// TwinCAT 3 PLC project MAIN
// ProgramVersion: 3.1.4024.0
// libraries:
//   CmpBitmapPool, * (System)
//   Tc2_Standard, * (Beckhoff Automation GmbH)
//   Tc2_System, * (Beckhoff Automation GmbH)
//   Tc3_IoLink, * (Beckhoff Automation GmbH)
//   Tc3_Module, * (Beckhoff Automation GmbH)
//   Util, * (System)
//   VisuSymbols,3.5.10.0,System
// project tree:
//   DUTs/ ImagePool.TcIPO (not stored)
//   / GlobalTextList.TcGTLO, PlcTask.TcTTO, Visualisierungsmanager.TcVMO (not stored), VISU_TASK.TcTTO
//   POUs/Grundfunktionen/ OID200DatenLesen.TcPOU, Hydr_Ventil.TcPOU
//   POUs/Unterfunktionen/ Ansteuerung_Ausgaenge.TcPOU, Automatik_Betrieb.TcPOU, Manueller_Betrieb.TcPOU, Meldeleuchte.TcPOU, Referenzfahrt.TcPOU, Warmlauf.TcPOU
//   POUs/ Saegeautomat.TcPOU, MAIN.TcPOU
//   VISUs/ Visualization.TcVIS
// real-time tasks:
//   TASK PlcTask: cycle T#10ms, priority 20, ADS port 350
//   TASK VISU_TASK: cycle T#200000us, priority 30, ADS port 351
// I/O:
//   DEVICE Gerät 5 (EtherCAT), AmsNetId 5.93.150.74.6.1
//     Klemme 2 (EK1100) [EK1100 EtherCAT-Koppler (2A E-Bus)]
//       Klemme 3 (EL6224) [EL6224 (IO Link Master)]
//       Klemme 4 (EL2024) [EL2024 4K. Dig. Ausgang 24V, 2A]
//       Klemme 5 (EL2024) [EL2024 4K. Dig. Ausgang 24V, 2A]
//       Klemme 5 (EL9011) [EL9011 Endklemme]
//   DEVICE Gerät 7 (CX-BK)
//     Box 1 (CX-BK)
// variable links:
//   MAIN/MAIN Instance <-> Device 5 (EtherCAT)/Term 2 (EK1100)/Term 3 (EL6224)
//     PlcTask Inputs/MAIN.Saegeautomat.OID200.ProzessDatenOID200 <-> IO-Link Port1/Port1: process data
//   MAIN/MAIN Instance <-> Device 5 (EtherCAT)/Term 2 (EK1100)/Term 4 (EL2024)
//     PlcTask Outputs/MAIN.Saegeautomat.Ansteuerung_Ausgaenge.OUT_Stammklemmung_Oben_Hoch <-> Channel 1/Output
//     PlcTask Outputs/MAIN.Saegeautomat.Ansteuerung_Ausgaenge.OUT_Stammklemmung_Oben_Runter <-> Channel 2/Output
//     PlcTask Outputs/MAIN.Saegeautomat.Ansteuerung_Ausgaenge.OUT_Stammklemmung_Unten_Hoch <-> Channel 3/Output
//     PlcTask Outputs/MAIN.Saegeautomat.Ansteuerung_Ausgaenge.OUT_Stammklemmung_Unten_Runter <-> Channel 4/Output
//   MAIN/MAIN Instance <-> Device 5 (EtherCAT)/Term 2 (EK1100)/Term 5 (EL2024)
//     PlcTask Outputs/MAIN.Saegeautomat.Ansteuerung_Ausgaenge.OUT_Saege_Heben <-> Channel 1/Output
//     PlcTask Outputs/MAIN.Saegeautomat.Ansteuerung_Ausgaenge.OUT_Saege_Senken <-> Channel 2/Output
//     PlcTask Outputs/MAIN.Saegeautomat.Ansteuerung_Ausgaenge.OUT_Stammklemmung_Unten_Runter <-> Channel 3/Output
//   MAIN/MAIN Instance <-> Device 7 (CX-BK)/Box 1 (CX-BK)
//     PlcTask Inputs/MAIN.Saegeautomat.IN_BetriebsArt_Automatik <-> Term 2 (KL1104)/Channel 3/Eingang
//     PlcTask Inputs/MAIN.Saegeautomat.IN_BetriebsArt_Manuell <-> Term 2 (KL1104)/Channel 4/Eingang
//     PlcTask Inputs/MAIN.Saegeautomat.IN_BetriebsArt_Referenz <-> Term 2 (KL1104)/Channel 1/Eingang
//     PlcTask Inputs/MAIN.Saegeautomat.IN_BetriebsArt_Warmlauf <-> Term 2 (KL1104)/Channel 2/Eingang
//     PlcTask Inputs/MAIN.Saegeautomat.IN_Einfache_Klemmung <-> Term 3 (KL1104)/Channel 4/Eingang
//     PlcTask Inputs/MAIN.Saegeautomat.IN_Endl_Obere_Stammklemmung_Oben <-> Term 7 (KL1104)/Channel 1/Eingang
//     PlcTask Inputs/MAIN.Saegeautomat.IN_Endl_Obere_Stammklemmung_Unten <-> Term 7 (KL1104)/Channel 2/Eingang
//     PlcTask Inputs/MAIN.Saegeautomat.IN_Endl_Saege_Oben <-> Term 8 (KL1104)/Channel 1/Eingang
//     PlcTask Inputs/MAIN.Saegeautomat.IN_Endl_Saege_Unten <-> Term 8 (KL1104)/Channel 2/Eingang
//     PlcTask Inputs/MAIN.Saegeautomat.IN_Endl_Tastschiene <-> Term 9 (KL1104)/Channel 3/Eingang
//     PlcTask Inputs/MAIN.Saegeautomat.IN_Endl_Untere_Stammklemmung_Oben <-> Term 7 (KL1104)/Channel 3/Eingang
//     PlcTask Inputs/MAIN.Saegeautomat.IN_Endl_Untere_Stammklemmung_Unten <-> Term 7 (KL1104)/Channel 4/Eingang
//     PlcTask Inputs/MAIN.Saegeautomat.IN_Endl_Zufuehrer_Hinten <-> Term 9 (KL1104)/Channel 1/Eingang
//     PlcTask Inputs/MAIN.Saegeautomat.IN_Endl_Zufuehrer_Vorne <-> Term 8 (KL1104)/Channel 4/Eingang
//     PlcTask Inputs/MAIN.Saegeautomat.IN_Hydraulik_EIN <-> Term 4 (KL1104)/Channel 2/Eingang
//     PlcTask Inputs/MAIN.Saegeautomat.IN_Kettenoel_nicht_Leer <-> Term 6 (KL1104)/Channel 3/Eingang
//     PlcTask Inputs/MAIN.Saegeautomat.IN_Kettenschmierung_Manuell_EIN <-> Term 6 (KL1104)/Channel 4/Eingang
//     PlcTask Inputs/MAIN.Saegeautomat.IN_Programm_Einzelsatz <-> Term 3 (KL1104)/Channel 3/Eingang
//     PlcTask Inputs/MAIN.Saegeautomat.IN_Saege_EIN <-> Term 4 (KL1104)/Channel 1/Eingang
//     PlcTask Inputs/MAIN.Saegeautomat.IN_Saege_Hoch <-> Term 6 (KL1104)/Channel 1/Eingang
//     PlcTask Inputs/MAIN.Saegeautomat.IN_Saege_Runter <-> Term 6 (KL1104)/Channel 2/Eingang
//     PlcTask Inputs/MAIN.Saegeautomat.IN_Schaltausg_Druckschalter_Obere_Klemmung <-> Term 9 (KL1104)/Channel 2/Eingang
//     PlcTask Inputs/MAIN.Saegeautomat.IN_Schaltausg_Lichtschranke <-> Term 9 (KL1104)/Channel 4/Eingang
//     PlcTask Inputs/MAIN.Saegeautomat.IN_Stammklemmer_Oben_Hoch <-> Term 5 (KL1104)/Channel 1/Eingang
//     PlcTask Inputs/MAIN.Saegeautomat.IN_Stammklemmer_Oben_Runter <-> Term 5 (KL1104)/Channel 2/Eingang
//     PlcTask Inputs/MAIN.Saegeautomat.IN_Stammklemmer_Unten_Hoch <-> Term 5 (KL1104)/Channel 3/Eingang
//     PlcTask Inputs/MAIN.Saegeautomat.IN_Stammklemmer_Unten_Runter <-> Term 5 (KL1104)/Channel 4/Eingang
//     PlcTask Inputs/MAIN.Saegeautomat.IN_Vorposition_Zufuehrer <-> Term 8 (KL1104)/Channel 3/Eingang
//     PlcTask Inputs/MAIN.Saegeautomat.IN_Zufuehrer_Rueck <-> Term 4 (KL1104)/Channel 3/Eingang
//     PlcTask Inputs/MAIN.Saegeautomat.IN_Zufuehrer_Vor <-> Term 4 (KL1104)/Channel 4/Eingang
//     PlcTask Inputs/MAIN.Saegeautomat.IN_Zyklus_Start <-> Term 3 (KL1104)/Channel 1/Eingang
//     PlcTask Inputs/MAIN.Saegeautomat.IN_Zyklus_Stopp <-> Term 3 (KL1104)/Channel 2/Eingang
//     PlcTask Outputs/MAIN.Saegeautomat.Ansteuerung_Ausgaenge.OUT_Kettenschmierung_EIN <-> Term 11 (KL2114)/Channel 1/Ausgang
//     PlcTask Outputs/MAIN.Saegeautomat.Ansteuerung_Ausgaenge.OUT_Saege_EIN <-> Term 12 (KL2114)/Channel 2/Ausgang
//     PlcTask Outputs/MAIN.Saegeautomat.Ansteuerung_Ausgaenge.OUT_Zufuehrer_Antrieb_Rueck <-> Term 10 (KL2114)/Channel 4/Ausgang
//     PlcTask Outputs/MAIN.Saegeautomat.Ansteuerung_Ausgaenge.OUT_Zufuehrer_Antrieb_Vor <-> Term 10 (KL2114)/Channel 3/Ausgang
//     PlcTask Outputs/MAIN.Saegeautomat.OUT_Hydraulikpumpe_EIN <-> Term 10 (KL2114)/Channel 1/Ausgang
//     PlcTask Outputs/MAIN.Saegeautomat.Steuerung_Meldeleuchten.OUT_Meldeleuchte_Gelb <-> Term 11 (KL2114)/Channel 2/Ausgang
//     PlcTask Outputs/MAIN.Saegeautomat.Steuerung_Meldeleuchten.OUT_Meldeleuchte_Gruen <-> Term 11 (KL2114)/Channel 4/Ausgang
//     PlcTask Outputs/MAIN.Saegeautomat.Steuerung_Meldeleuchten.OUT_Meldeleuchte_Rot <-> Term 11 (KL2114)/Channel 3/Ausgang

CONFIGURATION MAIN
    RESOURCE PLC ON TwinCAT3
        TASK PlcTask(INTERVAL := T#10ms, PRIORITY := 20);
        TASK VISU_TASK(INTERVAL := T#200000us, PRIORITY := 30);
        PROGRAM MAIN WITH PlcTask : MAIN;
        PROGRAM VisuElems_Visu_Prg WITH VISU_TASK : VisuElems.Visu_Prg;
    END_RESOURCE
END_CONFIGURATION

// ---- POUs/MAIN.TcPOU
PROGRAM MAIN
VAR
	Saegeautomat : Saegeautomat;
END_VAR

Saegeautomat();

END_PROGRAM

// ---- POUs/Saegeautomat.TcPOU
FUNCTION_BLOCK Saegeautomat
VAR_INPUT
END_VAR
VAR_OUTPUT
END_VAR
VAR
	//Eingänge Bedienung
	//Organisatorisches
	IN_BetriebsArt_Referenz AT %I* : BOOL;
	IN_BetriebsArt_Warmlauf AT %I* : BOOL;
	IN_BetriebsArt_Automatik AT %I* : BOOL;
	IN_BetriebsArt_Manuell AT %I* : BOOL;
	IN_Kein_Notaus AT %I* : BOOL := TRUE;
	IN_Maschine_EIN AT %I* : BOOL := TRUE;
	IN_Hydraulik_EIN AT %I* : BOOL;
	IN_Maschine_AUS AT %I* : BOOL;
	IN_Hydraulik_AUS AT %I* : BOOL;
	//Manuelle Bedienung
	IN_Kettenschmierung_Manuell_EIN AT %I* : BOOL;
	IN_Zufuehrer_Vor AT %I* : BOOL;
	IN_Zufuehrer_Rueck AT %I* : BOOL;
	IN_Stammklemmer_Oben_Hoch AT %I* : BOOL;
	IN_Stammklemmer_Oben_Runter AT %I* : BOOL;
	IN_Stammklemmer_Unten_Hoch AT %I* : BOOL;
	IN_Stammklemmer_Unten_Runter AT %I* : BOOL;
	IN_Saege_EIN AT %I* : BOOL;
	IN_Saege_AUS AT %I* : BOOL;
	IN_Saege_Hoch AT %I* : BOOL;
	IN_Saege_Runter AT %I* : BOOL;
	//Automatikmodus
	IN_Programm_Einzelsatz AT %I* : BOOL;
	IN_Zyklus_Start AT %I* : BOOL;
	IN_Zyklus_Stopp AT %I* : BOOL;
	IN_Einfache_Klemmung AT %I* : BOOL;
	
	
	//Eingänge Sensorik
	//Zuführer
	IN_Endl_Zufuehrer_Hinten AT %I* : BOOL;
	IN_Endl_Zufuehrer_Vorne AT %I* : BOOL;
	IN_Vorposition_Zufuehrer AT %I* : BOOL;
	IOL_Schaltausg_Distanzsensor_Holzende : BOOL; //Über Schaltausgang oder IO-Link Analogdaten?
	IOL_DistanzSensor_Abst : UINT;
	IN_Schaltausg_Lichtschranke AT %I* : BOOL; 
	
	//Stammklemmung Oben
	IN_Endl_Obere_Stammklemmung_Oben AT %I* : BOOL;
	IN_Endl_Obere_Stammklemmung_Unten AT %I* : BOOL;
	IN_Endl_Tastschiene AT %I* : BOOL;
	IN_Schaltausg_Druckschalter_Obere_Klemmung AT %I* : BOOL;
	//Stammklemmung Unten
	IN_Endl_Untere_Stammklemmung_Oben AT %I* : BOOL;
	IN_Endl_Untere_Stammklemmung_Unten AT %I* : BOOL;
	//Säge
	IN_Endl_Saege_Oben AT %I* : BOOL;
	IN_Endl_Saege_Unten AT %I* : BOOL;
	IN_Kettenoel_nicht_Leer AT %I* : BOOL;
	
	//Ausgänge
	//Ausgänge Hydraulik
	
	//Ausgänge Schalten
	OUT_Hydraulikpumpe_EIN AT %Q* : BOOL;
	//Ausgänge Daten
	
	
		
		
	//Interne Merker
	Maschine_EIN : BOOL;
	Hydraulik_EIN : BOOL;
	Referenz_gefahren : BOOL;
	Zyklus_beendet : BOOL;
	busy : BOOL;
	warten : BOOL;
	
	
	Referenzfahrt : Referenzfahrt;
	Warmlauf : Warmlauf;
	Manueller_Betrieb : Manueller_Betrieb;
	Automatikbetrieb : Automatik_Betrieb;
	Steuerung_Meldeleuchten : Meldeleuchte;
	OID200 : OID200DatenLesen;
	Ansteuerung_Ausgaenge : Ansteuerung_Ausgaenge;
	
	P_Flanke_Zyklus_Stopp : R_TRIG;
	P_Flanke_Zyklus_Start : R_TRIG;
	P_Flanke_Maschine_EIN : R_TRIG;
	

	
END_VAR

P_Flanke_Zyklus_Stopp(CLK := NOT IN_Zyklus_Stopp);
P_Flanke_Zyklus_Start(CLK := IN_Zyklus_Start);
P_Flanke_Maschine_EIN(CLK := IN_Maschine_EIN);


IF IN_Kein_Notaus AND IN_Maschine_EIN THEN
	Maschine_EIN := TRUE;
ELSIF NOT IN_Kein_Notaus OR IN_Maschine_AUS THEN
	Maschine_EIN := FALSE;
END_IF

IF Maschine_EIN AND IN_BetriebsArt_Referenz THEN
	Referenzfahrt(
		Kein_Notaus := IN_Kein_Notaus,
		Programm_Einzelsatz := IN_Programm_Einzelsatz,
		Zyklus_Start := P_Flanke_Zyklus_Start.Q,
		SFCInit := P_Flanke_Zyklus_Stopp.Q OR NOT IN_Kein_Notaus,
		SFCTipMode := IN_Programm_Einzelsatz,
		SFCTip := P_Flanke_Zyklus_Start.Q,
		Endl_Saege_Oben := NOT IN_Endl_Saege_Oben,
		Endl_Obere_Stammklemmung_Oben := NOT IN_Endl_Obere_Stammklemmung_Oben,
		Endl_Untere_Stammklemmung_Unten := NOT IN_Endl_Untere_Stammklemmung_Unten,
		Endl_Zufuehrer_Hinten := NOT IN_Endl_Zufuehrer_Hinten,
		busy := busy,
		Referenz_Gefahren := Referenz_gefahren,
		Zyklus_Beendet := Zyklus_beendet);	
END_IF

IF Maschine_EIN AND IN_BetriebsArt_Warmlauf THEN
	Warmlauf();
END_IF

IF Maschine_EIN AND IN_BetriebsArt_Manuell THEN
	Manueller_Betrieb(
		Kein_Notaus:= IN_Kein_Notaus, 
		Hydraulik_EIN:= IN_Hydraulik_EIN, 
		Hydraulik_AUS:= IN_Hydraulik_AUS, 
		Kettenschmierung_Manuell_EIN:= IN_Kettenschmierung_Manuell_EIN, 
		Zufuehrer_Vor:= IN_Zufuehrer_Vor, 
		Zufuehrer_Rueck:= IN_Zufuehrer_Rueck, 
		Stammklemmer_Oben_Hoch:= IN_Stammklemmer_Oben_Hoch, 
		Stammklemmer_Oben_Runter:= IN_Stammklemmer_Oben_Runter, 
		Stammklemmer_Unten_Hoch:= IN_Stammklemmer_Unten_Hoch, 
		Stammklemmer_Unten_Runter:= IN_Stammklemmer_Unten_Runter, 
		Saege_EIN:= IN_Saege_EIN, 
		Saege_AUS:= IN_Saege_AUS, 
		Saege_Hoch:= IN_Saege_Hoch, 
		Saege_Runter:= IN_Saege_Runter, 
		Endl_Zufuehrer_Hinten:= NOT IN_Endl_Zufuehrer_Hinten, 
		Endl_Zufuehrer_Vorne:= NOT IN_Endl_Zufuehrer_Vorne, 
		Vorposition_Zufuehrer:= NOT IN_Vorposition_Zufuehrer,  
		Endl_Obere_Stammklemmung_Oben:= NOT IN_Endl_Obere_Stammklemmung_Oben, 
		Endl_Obere_Stammklemmung_Unten:= NOT IN_Endl_Obere_Stammklemmung_Unten, 
		Endl_Tastschiene:= NOT IN_Endl_Tastschiene, 
		Schaltausg_Druckschalter_Obere_Klemmung:= NOT IN_Schaltausg_Druckschalter_Obere_Klemmung, 
		Endl_Untere_Stammklemmung_Oben:= NOT IN_Endl_Untere_Stammklemmung_Oben, 
		Endl_Untere_Stammklemmung_Unten:= NOT IN_Endl_Untere_Stammklemmung_Unten, 
		Endl_Saege_Oben:= NOT IN_Endl_Saege_Oben, 
		Endl_Saege_Unten:= NOT IN_Endl_Saege_Unten, 
		);
	
END_IF

IF Maschine_EIN AND IN_BetriebsArt_Automatik THEN
	Automatikbetrieb(
	Kein_Notaus:= IN_Kein_Notaus, 
	Zyklus_Start:= IN_Zyklus_Start, 
	Zyklus_Stopp:= NOT IN_Zyklus_Stopp, 
	Einfache_Klemmung := IN_Einfache_Klemmung,
	SFCInit:= not IN_Zyklus_Stopp, 
	SFCTip:= IN_Programm_Einzelsatz AND IN_Zyklus_Start, 
	SFCTipMode:= IN_Programm_Einzelsatz, 
	Endl_Zufuehrer_Hinten:= NOT IN_Endl_Zufuehrer_Hinten, 
	Endl_Zufuehrer_Vorne:= NOT IN_Endl_Zufuehrer_Vorne, 
	Vorposition_Zufuehrer:= NOT IN_Vorposition_Zufuehrer, 
	IOL_Schaltausg_Distanzsensor_Holzende:= NOT IN_Schaltausg_Lichtschranke, 
	IOL_DistanzSensor_Abst:= IOL_DistanzSensor_Abst, 
	Endl_Obere_Stammklemmung_Oben:= NOT IN_Endl_Obere_Stammklemmung_Oben, 
	Endl_Obere_Stammklemmung_Unten:= NOT IN_Endl_Obere_Stammklemmung_Unten, 
	Endl_Tastschiene:= IN_Endl_Tastschiene, 
	Schaltausg_Druckschalter_Obere_Klemmung:= not IN_Schaltausg_Druckschalter_Obere_Klemmung, 
	Endl_Untere_Stammklemmung_Oben:= NOT IN_Endl_Untere_Stammklemmung_Oben, 
	Endl_Untere_Stammklemmung_Unten:= NOT IN_Endl_Untere_Stammklemmung_Unten, 
	Endl_Saege_Oben:= NOT IN_Endl_Saege_Oben, 
	Endl_Saege_Unten:= NOT IN_Endl_Saege_Unten, 
	Warten_Auf_Weiterschalten=> , 
	Warten_auf_Material=> , 
	QStammklemmung_Oben_Hoch=> , 
	QStammklemmung_Oben_Runter=> , 
	QStammklemmung_Unten_Hoch=> , 
	QStammklemmung_Unten_Runter=> , 
	QSaege_Senken=> , 
	QSaege_Heben=> , 
	QHydraulikpumpe_EIN=> , 
	QZufuehrer_Antrieb_vor=> , 
	QZufuehrer_Antrieb_Rueck=> , 
	QSaege_Antrieb_Ein=> , 
	QKettenschmierung_EIN=> , 
	warten:= warten, 
	Hydraulik_EIN:= Hydraulik_EIN, 
	Zyklus_Beendet:= Zyklus_beendet);
END_IF

Ansteuerung_Ausgaenge(
	Saege_Hoch:= Referenzfahrt.Saege_Heben OR Manueller_Betrieb.QSaege_Heben OR Automatikbetrieb.QSaege_Heben, 
	Saege_Runter:= Manueller_Betrieb.QSaege_Senken OR Automatikbetrieb.QSaege_Senken, 
	Stammklemmung_Oben_Hoch:= Referenzfahrt.Stammklemmung_oben_Hoch OR Manueller_Betrieb.QStammklemmung_Oben_Hoch OR Automatikbetrieb.QStammklemmung_Oben_Hoch, 
	Stammklemmung_Oben_Runter:= Manueller_Betrieb.QStammklemmung_Oben_Runter OR Automatikbetrieb.QStammklemmung_Oben_Runter, 
	Stammklemmung_Unten_Hoch:= Manueller_Betrieb.QStammklemmung_Unten_Hoch OR Automatikbetrieb.QStammklemmung_Unten_Hoch,
	Stammklemmung_Unten_Runter:= Referenzfahrt.Stammklemmung_unten_Runter OR Manueller_Betrieb.QStammklemmung_Unten_Runter OR Automatikbetrieb.QStammklemmung_Unten_Runter,
	Saege_EIN := Manueller_Betrieb.QSaege_Antrieb_Ein OR Automatikbetrieb.QSaege_Antrieb_Ein,
	Zufuehrer_Vor := Manueller_Betrieb.QZufuehrer_Antrieb_vor OR Automatikbetrieb.QZufuehrer_Antrieb_vor,
	Zufuehrer_Rueck := Referenzfahrt.Zufuehrer_Zurueck OR Manueller_Betrieb.QZufuehrer_Antrieb_Rueck OR Automatikbetrieb.QZufuehrer_Antrieb_Rueck,
	endl_Zufuehrer_vorne := NOT IN_Endl_Zufuehrer_Vorne,
	endl_Zufuehrer_hinten := NOT IN_Endl_Zufuehrer_Hinten,
	endl_Zufuehrer_Vorpos := NOT IN_Vorposition_Zufuehrer,
	endl_Stammklemmung_Oben_Oben := NOT IN_Endl_Obere_Stammklemmung_Oben,
	endl_Stammklemmung_Oben_Unten := NOT IN_Endl_Obere_Stammklemmung_Unten,
	endl_Stammklemmung_Unten_Oben := NOT IN_Endl_Untere_Stammklemmung_Oben,
	endl_Stammklemmung_Unten_Unten := NOT IN_Endl_Untere_Stammklemmung_Unten,
	endl_Saege_Oben := NOT IN_Endl_Saege_Oben,
	endl_Saege_Unten:= NOT IN_Endl_Saege_Unten,
	kettenschmierung_EIN := Manueller_Betrieb.QKettenschmierung_EIN OR Automatikbetrieb.QSaege_Antrieb_Ein
);

OUT_Hydraulikpumpe_EIN := Manueller_Betrieb.QHydraulikpumpe_EIN OR Automatikbetrieb.QHydraulikpumpe_EIN OR Referenzfahrt.QHydraulik_EIN;

Steuerung_Meldeleuchten(
	Maschine_EIN := Maschine_EIN,
	Referenz_gefahren := Referenz_gefahren,
	Kettenschmierung_nicht_leer := IN_Kettenoel_nicht_Leer,
	Fehler_liegt_an := ,
	Busy := busy,
	Warten_auf_weiterschalten := Referenzfahrt.Warten_Auf_Weiterschalten OR FALSE, //Automatikbetrieb.Warten_Auf_Weiterschalten
	Zyklus_beendet := );


OID200(
 OID200SchaltSignal => IOL_Schaltausg_Distanzsensor_Holzende,
iOID200Dist_zu_Holz => IOL_DistanzSensor_Abst);

END_FUNCTION_BLOCK

// ---- POUs/Unterfunktionen/Referenzfahrt.TcPOU
FUNCTION_BLOCK Referenzfahrt
VAR_INPUT
	//Taster
	Kein_Notaus : BOOL;
	Programm_Einzelsatz : BOOL;
	Zyklus_Start : BOOL;
	Zyklus_Stopp : BOOL;
	//Merker
	SFCInit : BOOL;
	SFCTip : BOOL;
	SFCTipMode : BOOL;
	//Sensoren	
	Endl_Saege_Oben : BOOL;
	Endl_Obere_Stammklemmung_Oben : BOOL;
	Endl_Untere_Stammklemmung_Unten : BOOL;
	Endl_Zufuehrer_Hinten : BOOL;
	
END_VAR
VAR_OUTPUT
	Saege_Heben : BOOL;
	Stammklemmung_oben_Hoch : BOOL;
	Stammklemmung_unten_Runter : BOOL;
	Zufuehrer_Zurueck : BOOL;
	Warten_Auf_Weiterschalten : BOOL;
	QHydraulik_EIN : BOOL;

END_VAR
VAR_IN_OUT
	//Merker
	busy : BOOL;
	
	Referenz_Gefahren : BOOL;
	Zyklus_Beendet : BOOL;
	
END_VAR
VAR
END_VAR

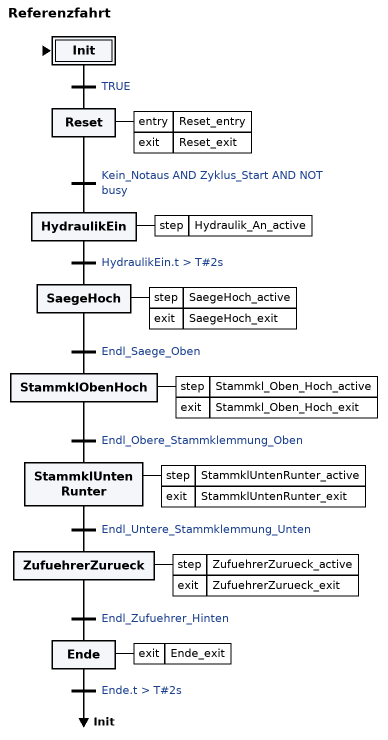
INITIAL_STEP Init:
END_STEP
TRANSITION FROM Init TO Reset
    := TRUE;
END_TRANSITION
STEP Reset:
    Reset_entry(P1);  // entry action
    Reset_exit(P0);  // exit action
END_STEP
TRANSITION FROM Reset TO HydraulikEin
    := Kein_Notaus AND Zyklus_Start AND NOT busy;
END_TRANSITION
STEP HydraulikEin:
    Hydraulik_An_active(N);  // step action
END_STEP
TRANSITION FROM HydraulikEin TO SaegeHoch
    := HydraulikEin.t > T#2s;
END_TRANSITION
STEP SaegeHoch:
    SaegeHoch_active(N);  // step action
    SaegeHoch_exit(P0);  // exit action
END_STEP
TRANSITION FROM SaegeHoch TO StammklObenHoch
    := Endl_Saege_Oben;
END_TRANSITION
STEP StammklObenHoch:
    Stammkl_Oben_Hoch_active(N);  // step action
    Stammkl_Oben_Hoch_exit(P0);  // exit action
END_STEP
TRANSITION FROM StammklObenHoch TO StammklUntenRunter
    := Endl_Obere_Stammklemmung_Oben;
END_TRANSITION
STEP StammklUntenRunter:
    StammklUntenRunter_active(N);  // step action
    StammklUntenRunter_exit(P0);  // exit action
END_STEP
TRANSITION FROM StammklUntenRunter TO ZufuehrerZurueck
    := Endl_Untere_Stammklemmung_Unten;
END_TRANSITION
STEP ZufuehrerZurueck:
    ZufuehrerZurueck_active(N);  // step action
    ZufuehrerZurueck_exit(P0);  // exit action
END_STEP
TRANSITION FROM ZufuehrerZurueck TO Ende
    := Endl_Zufuehrer_Hinten;
END_TRANSITION
STEP Ende:
    Ende_exit(P0);  // exit action
END_STEP
TRANSITION FROM Ende TO Init
    := Ende.t > T#2s;
END_TRANSITION

ACTION Abschluss_active:

END_ACTION

ACTION Ende_exit:
QHydraulik_EIN := FALSE;

busy := FALSE;
Referenz_Gefahren := TRUE;
Zyklus_Beendet := TRUE;
END_ACTION

ACTION Hydraulik_An_active:
QHydraulik_EIN := TRUE;

IF Kein_Notaus AND Zyklus_Start AND NOT busy AND Programm_Einzelsatz THEN 
	Warten_Auf_Weiterschalten := TRUE;
END_IF
END_ACTION

ACTION Hydraulik_An_exit:

END_ACTION

ACTION Reset_entry:
busy := FALSE;
QHydraulik_EIN := FALSE;
Saege_Heben := FALSE;
Stammklemmung_oben_Hoch := FALSE;
Stammklemmung_unten_Runter := FALSE;
Zufuehrer_Zurueck := FALSE;
END_ACTION

ACTION Reset_exit:
busy := TRUE;
Referenz_Gefahren := FALSE;
Zyklus_Beendet := FALSE;

Saege_Heben := FALSE;
Stammklemmung_oben_Hoch := FALSE;
Stammklemmung_unten_Runter := FALSE;
Zufuehrer_Zurueck := FALSE;
END_ACTION

ACTION SaegeHoch_active:
IF NOT Endl_Saege_Oben THEN
	Saege_Heben := TRUE;
END_IF
END_ACTION

ACTION SaegeHoch_exit:
Saege_Heben := FALSE;
END_ACTION

ACTION Stammkl_Oben_Hoch_active:
IF NOT Endl_Obere_Stammklemmung_Oben THEN
	Stammklemmung_oben_Hoch := TRUE;
END_IF
END_ACTION

ACTION Stammkl_Oben_Hoch_exit:
Stammklemmung_oben_Hoch := FALSE;
END_ACTION

ACTION StammklUntenRunter_active:
IF NOT Endl_Untere_Stammklemmung_Unten THEN
	Stammklemmung_unten_Runter := TRUE;
END_IF
END_ACTION

ACTION StammklUntenRunter_exit:
Stammklemmung_unten_Runter := False;
END_ACTION

ACTION ZufuehrerZurueck_active:
IF NOT Endl_Zufuehrer_Hinten THEN
	Zufuehrer_Zurueck := TRUE;
END_IF
END_ACTION

ACTION ZufuehrerZurueck_exit:
Zufuehrer_Zurueck := FALSE;
END_ACTION

END_FUNCTION_BLOCK

// ---- POUs/Unterfunktionen/Warmlauf.TcPOU
FUNCTION_BLOCK Warmlauf
VAR_INPUT
END_VAR
VAR_OUTPUT
END_VAR
VAR
	
END_VAR

END_FUNCTION_BLOCK

// ---- POUs/Unterfunktionen/Manueller_Betrieb.TcPOU
FUNCTION_BLOCK Manueller_Betrieb
VAR_INPUT
	Kein_Notaus : BOOL;
	//Taster auf Bedienfeld
	Hydraulik_EIN : BOOL;
	Hydraulik_AUS : BOOL;
	Kettenschmierung_Manuell_EIN : BOOL;
	Zufuehrer_Vor : BOOL;
	Zufuehrer_Rueck : BOOL;
	Stammklemmer_Oben_Hoch : BOOL;
	Stammklemmer_Oben_Runter : BOOL;
	Stammklemmer_Unten_Hoch : BOOL;
	Stammklemmer_Unten_Runter : BOOL;
	Saege_EIN : BOOL;
	Saege_AUS : BOOL;
	Saege_Hoch : BOOL;
	Saege_Runter : BOOL;
	
	
	//Eingänge Sensorik
	//Zuführer
	Endl_Zufuehrer_Hinten : BOOL;
	Endl_Zufuehrer_Vorne : BOOL;
	Vorposition_Zufuehrer : BOOL;
	//Stammklemmung Oben
	Endl_Obere_Stammklemmung_Oben : BOOL;
	Endl_Obere_Stammklemmung_Unten : BOOL;
	Endl_Tastschiene : BOOL;
	Schaltausg_Druckschalter_Obere_Klemmung : BOOL;
	//Stammklemmung Unten
	Endl_Untere_Stammklemmung_Oben : BOOL;
	Endl_Untere_Stammklemmung_Unten : BOOL;
	//Säge
	Endl_Saege_Oben : BOOL;
	Endl_Saege_Unten : BOOL;
END_VAR
VAR_OUTPUT
	//Ausgänge Hydraulik
	QStammklemmung_Oben_Hoch : BOOL;
	QStammklemmung_Oben_Runter : BOOL;
	QStammklemmung_Unten_Hoch : BOOL;
	QStammklemmung_Unten_Runter : BOOL;
	QSaege_Senken : BOOL;
	QSaege_Heben : BOOL;
	//Ausgänge Schalten
	QHydraulikpumpe_EIN : BOOL;
	QZufuehrer_Antrieb_vor : BOOL;
	QZufuehrer_Antrieb_Rueck : BOOL;
	QSaege_Antrieb_Ein : BOOL;
	QKettenschmierung_EIN : BOOL;
	//Ausgänge Daten
	//FU DATEN
END_VAR
VAR_IN_OUT
	
	
END_VAR
VAR
	Impulsgeber : BLINK;
	TON_Timer_Impuls : TON;
	TON_Timer_Pause : TON;
	Impuls_Zeit : TIME := T#3S;
	Pause_Zeit : TIME := T#3S;
	Impuls : BOOL;
END_VAR

QStammklemmung_Oben_Hoch :=
QStammklemmung_Oben_Runter := 
QStammklemmung_Unten_Hoch := 
QStammklemmung_Unten_Runter := 
QSaege_Senken := 
QSaege_Heben := 
QZufuehrer_Antrieb_vor := 
QZufuehrer_Antrieb_Rueck := 
QSaege_Antrieb_Ein := 
QKettenschmierung_EIN := FALSE;

QHydraulikpumpe_EIN := Hydraulik_EIN;

//Funktionen mit Hydraulik
IF QHydraulikpumpe_EIN THEN
	QStammklemmung_Oben_Hoch := Stammklemmer_Oben_Hoch AND NOT Stammklemmer_Oben_Runter;
	QStammklemmung_Oben_Runter := Stammklemmer_Oben_Runter AND NOT Stammklemmer_Oben_Hoch;
	QStammklemmung_Unten_Hoch := Stammklemmer_Unten_Hoch AND NOT Stammklemmer_Unten_Runter;
	QStammklemmung_Unten_Runter := Stammklemmer_Unten_Runter AND NOT Stammklemmer_Unten_Hoch;
	QSaege_Senken := Saege_Runter AND NOT Saege_Hoch AND NOT Saege_Hoch;
	QSaege_Heben := Saege_Hoch AND NOT Saege_Runter AND NOT Saege_Runter;
END_IF

//Funktionen ohne Hydraulik
IF Hydraulik_EIN THEN
	QHydraulikpumpe_EIN := TRUE;
ELSIF Hydraulik_AUS THEN
	QHydraulikpumpe_EIN := FALSE;
END_IF

QZufuehrer_Antrieb_vor := Zufuehrer_Vor AND NOT Zufuehrer_Rueck;
QZufuehrer_Antrieb_Rueck := Zufuehrer_Rueck AND NOT Zufuehrer_Vor;

QSaege_Antrieb_Ein := Saege_EIN;

Impulsgeber(
	ENABLE := Kettenschmierung_Manuell_EIN,
	TIMELOW := Pause_Zeit,
	TIMEHIGH := Impuls_Zeit,
	OUT => Impuls);

QKettenschmierung_EIN := Kettenschmierung_Manuell_EIN AND Impuls;

END_FUNCTION_BLOCK

// ---- POUs/Unterfunktionen/Automatik_Betrieb.TcPOU
FUNCTION_BLOCK Automatik_Betrieb
VAR_INPUT
	Kein_Notaus : BOOL;
	Zyklus_Start : BOOL;
	Zyklus_Stopp : BOOL;
	SFCInit : BOOL;
	SFCTip : BOOL;
	SFCTipMode : BOOL;
	Einfache_Klemmung : BOOL;
	
	//Eingänge Sensorik
	//Zuführer
	Endl_Zufuehrer_Hinten : BOOL;
	Endl_Zufuehrer_Vorne : BOOL;
	Vorposition_Zufuehrer : BOOL;
	IOL_Schaltausg_Distanzsensor_Holzende : BOOL; //Über Schaltausgang oder IO-Link Analogdaten?
	IOL_DistanzSensor_Abst : UINT;
	//Stammklemmung Oben
	Endl_Obere_Stammklemmung_Oben : BOOL;
	Endl_Obere_Stammklemmung_Unten : BOOL;
	Endl_Tastschiene : BOOL;
	Schaltausg_Druckschalter_Obere_Klemmung : BOOL;
	//Stammklemmung Unten
	Endl_Untere_Stammklemmung_Oben : BOOL;
	Endl_Untere_Stammklemmung_Unten : BOOL;
	//Säge
	Endl_Saege_Oben : BOOL;
	Endl_Saege_Unten : BOOL;
	
END_VAR
VAR_OUTPUT
	Warten_Auf_Weiterschalten :BOOL;
	Warten_auf_Material : BOOL;
	//Hydraulik
	QStammklemmung_Oben_Hoch : BOOL;
	QStammklemmung_Oben_Runter : BOOL;
	QStammklemmung_Unten_Hoch : BOOL;
	QStammklemmung_Unten_Runter : BOOL;
	QSaege_Senken : BOOL;
	QSaege_Heben : BOOL;
	//Ausgänge Schalten
	QHydraulikpumpe_EIN : BOOL;
	QZufuehrer_Antrieb_vor : BOOL;
	QZufuehrer_Antrieb_Rueck : BOOL;
	QSaege_Antrieb_Ein : BOOL;
	QKettenschmierung_EIN : BOOL;
	
END_VAR
VAR_IN_OUT
	warten : BOOL;
	Hydraulik_EIN : BOOL;
	Zyklus_Beendet : BOOL;
END_VAR
VAR
	Holz_Fertig : BOOL;
	Holz_Geklemmt : BOOL;
END_VAR

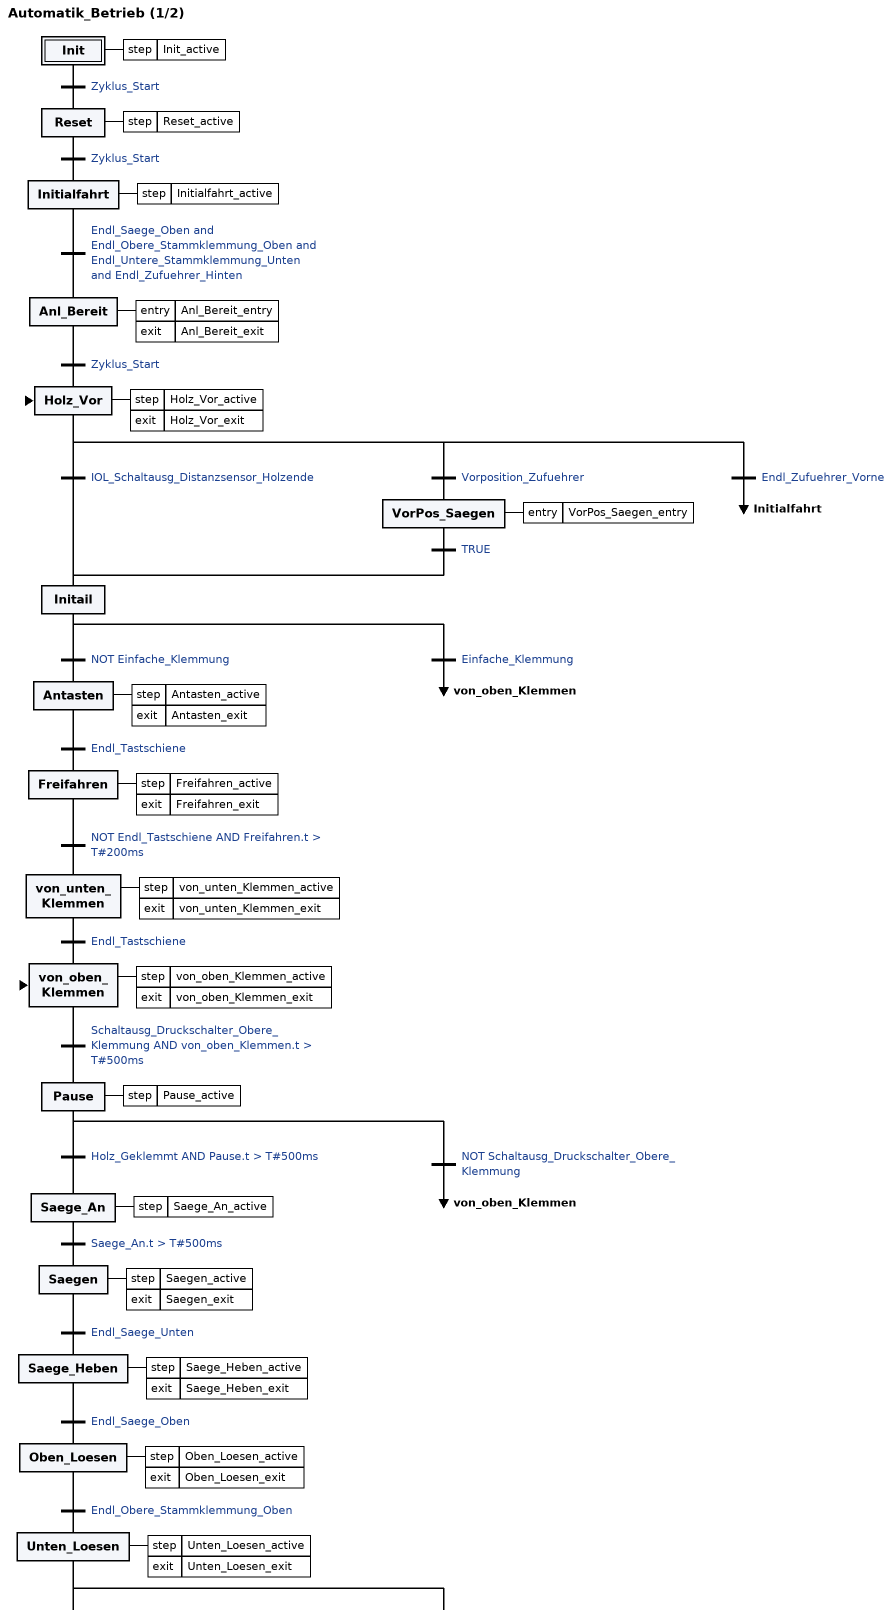
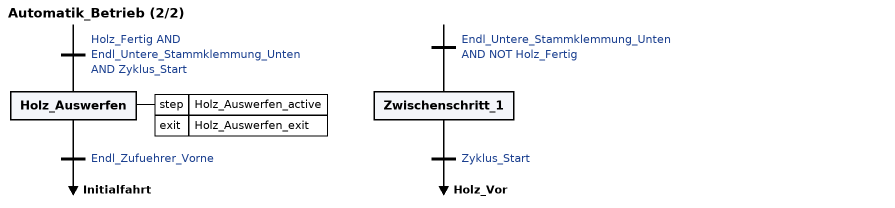
INITIAL_STEP Init:
    Init_active(N);  // step action
END_STEP
TRANSITION FROM Init TO Reset
    := Zyklus_Start;
END_TRANSITION
STEP Reset:
    Reset_active(N);  // step action
END_STEP
TRANSITION FROM Reset TO Initialfahrt_
    := Zyklus_Start;
END_TRANSITION
STEP Initialfahrt_:  // name as stored: Initialfahrt 
    Initialfahrt_active(N);  // step action
END_STEP
TRANSITION FROM Initialfahrt_ TO Anl_Bereit
    := Endl_Saege_Oben and Endl_Obere_Stammklemmung_Oben and Endl_Untere_Stammklemmung_Unten and Endl_Zufuehrer_Hinten;
END_TRANSITION
STEP Anl_Bereit:
    Anl_Bereit_entry(P1);  // entry action
    Anl_Bereit_exit(P0);  // exit action
END_STEP
TRANSITION FROM Anl_Bereit TO Holz_Vor
    := Zyklus_Start;
END_TRANSITION
STEP Holz_Vor:
    Holz_Vor_active(N);  // step action
    Holz_Vor_exit(P0);  // exit action
END_STEP
TRANSITION FROM Holz_Vor TO Initail
    := IOL_Schaltausg_Distanzsensor_Holzende;
END_TRANSITION
TRANSITION FROM Holz_Vor TO VorPos_Saegen
    := Vorposition_Zufuehrer;
END_TRANSITION
STEP VorPos_Saegen:
    VorPos_Saegen_entry(P1);  // entry action
END_STEP
TRANSITION FROM VorPos_Saegen TO Initail
    := TRUE;
END_TRANSITION
TRANSITION FROM Holz_Vor TO Initialfahrt
    := Endl_Zufuehrer_Vorne;
END_TRANSITION
// macro Holz_Klemmen begins
STEP Initail:
END_STEP
TRANSITION FROM Initail TO Antasten
    := NOT Einfache_Klemmung;
END_TRANSITION
STEP Antasten:
    Antasten_active(N);  // step action
    Antasten_exit(P0);  // exit action
END_STEP
TRANSITION FROM Initail TO von_oben_Klemmen
    := Einfache_Klemmung;
END_TRANSITION
TRANSITION FROM Antasten TO Freifahren
    := Endl_Tastschiene;
END_TRANSITION
STEP Freifahren:
    Freifahren_active(N);  // step action
    Freifahren_exit(P0);  // exit action
END_STEP
TRANSITION FROM Freifahren TO von_unten_Klemmen
    := NOT Endl_Tastschiene AND Freifahren.t > T#200ms;
END_TRANSITION
STEP von_unten_Klemmen:
    von_unten_Klemmen_active(N);  // step action
    von_unten_Klemmen_exit(P0);  // exit action
END_STEP
TRANSITION FROM von_unten_Klemmen TO von_oben_Klemmen
    := Endl_Tastschiene;
END_TRANSITION
STEP von_oben_Klemmen:
    von_oben_Klemmen_active(N);  // step action
    von_oben_Klemmen_exit(P0);  // exit action
END_STEP
TRANSITION FROM von_oben_Klemmen TO Pause
    := Schaltausg_Druckschalter_Obere_Klemmung AND von_oben_Klemmen.t > T#500ms;
END_TRANSITION
STEP Pause:
    Pause_active(N);  // step action
END_STEP
TRANSITION FROM Pause TO Saege_An
    := Holz_Geklemmt AND Pause.t > T#500ms;
END_TRANSITION
TRANSITION FROM Pause TO von_oben_Klemmen
    := NOT Schaltausg_Druckschalter_Obere_Klemmung;
END_TRANSITION
// macro Holz_Saegen begins
STEP Saege_An:
    Saege_An_active(N);  // step action
END_STEP
TRANSITION FROM Saege_An TO Saegen
    := Saege_An.t > T#500ms;
END_TRANSITION
STEP Saegen:
    Saegen_active(N);  // step action
    Saegen_exit(P0);  // exit action
END_STEP
TRANSITION FROM Saegen TO Saege_Heben
    := Endl_Saege_Unten;
END_TRANSITION
STEP Saege_Heben:
    Saege_Heben_active(N);  // step action
    Saege_Heben_exit(P0);  // exit action
END_STEP
TRANSITION FROM Saege_Heben TO Oben_Loesen
    := Endl_Saege_Oben;
END_TRANSITION
// macro Holz_Klemmung_Loesen begins
STEP Oben_Loesen:
    Oben_Loesen_active(N);  // step action
    Oben_Loesen_exit(P0);  // exit action
END_STEP
TRANSITION FROM Oben_Loesen TO Unten_Loesen
    := Endl_Obere_Stammklemmung_Oben;
END_TRANSITION
STEP Unten_Loesen:
    Unten_Loesen_active(N);  // step action
    Unten_Loesen_exit(P0);  // exit action
END_STEP
TRANSITION FROM Unten_Loesen TO Holz_Auswerfen
    := Holz_Fertig AND Endl_Untere_Stammklemmung_Unten AND Zyklus_Start;
END_TRANSITION
STEP Holz_Auswerfen:
    Holz_Auswerfen_active(N);  // step action
    Holz_Auswerfen_exit(P0);  // exit action
END_STEP
TRANSITION FROM Holz_Auswerfen TO Initialfahrt
    := Endl_Zufuehrer_Vorne;
END_TRANSITION
TRANSITION FROM Unten_Loesen TO Zwischenschritt_1
    := Endl_Untere_Stammklemmung_Unten AND NOT Holz_Fertig;
END_TRANSITION
STEP Zwischenschritt_1:
END_STEP
TRANSITION FROM Zwischenschritt_1 TO Holz_Vor
    := Zyklus_Start;
END_TRANSITION

ACTION Anl_Bereit_entry:
Warten_auf_Material := TRUE;
QHydraulikpumpe_EIN := FALSE;
END_ACTION

ACTION Anl_Bereit_exit:
Warten_auf_Material := FALSE;
QHydraulikpumpe_EIN := TRUE;
END_ACTION

ACTION Antasten_active:
QStammklemmung_Oben_Runter := TRUE;
END_ACTION

ACTION Antasten_exit:
QStammklemmung_Oben_Runter := FALSE;
END_ACTION

ACTION Freifahren_active:
QStammklemmung_Oben_Hoch := TRUE;
END_ACTION

ACTION Freifahren_exit:
QStammklemmung_Oben_Hoch := FALSE;
END_ACTION

ACTION Holz_Auswerfen_active:
QZufuehrer_Antrieb_vor := TRUE;
END_ACTION

ACTION Holz_Auswerfen_exit:
QZufuehrer_Antrieb_vor := FALSE;
Holz_Fertig := FALSE;
END_ACTION

ACTION Holz_Vor_active:
IF NOT Vorposition_Zufuehrer AND NOT Endl_Zufuehrer_Vorne THEN
	QZufuehrer_Antrieb_vor := TRUE;
END_IF 


IF Vorposition_Zufuehrer OR Endl_Zufuehrer_Vorne OR IOL_Schaltausg_Distanzsensor_Holzende THEN
	QZufuehrer_Antrieb_vor := FALSE;
END_IF
END_ACTION

ACTION Holz_Vor_exit:
QZufuehrer_Antrieb_vor := FALSE;
END_ACTION

ACTION Init_active:
QStammklemmung_Oben_Hoch := 
QStammklemmung_Oben_Runter := 
QStammklemmung_Unten_Hoch := 
QStammklemmung_Unten_Runter := 
QSaege_Senken := 
QSaege_Heben := 
//Ausgänge Schalten
QHydraulikpumpe_EIN := 
QZufuehrer_Antrieb_vor := 
QZufuehrer_Antrieb_Rueck := 
QSaege_Antrieb_Ein := 
QKettenschmierung_EIN := 
Warten_Auf_Weiterschalten :=
Zyklus_Beendet := FALSE;
END_ACTION

ACTION Initialfahrt_active:
IF NOT Endl_Saege_Oben THEN
	QSaege_Heben := TRUE;
	warten := TRUE;
ELSE 
	QSaege_Heben := FALSE;
	warten := FALSE;
END_IF

IF NOT Endl_Obere_Stammklemmung_Oben AND NOT warten THEN
	QStammklemmung_Oben_Hoch := TRUE;
	warten := TRUE;
ELSE
	QStammklemmung_Oben_Hoch := FALSE;
	warten := FALSE;
END_IF

IF NOT Endl_Untere_Stammklemmung_Unten AND NOT warten THEN 
	QStammklemmung_Unten_Runter := TRUE;
	warten := TRUE;
ELSE 
	QStammklemmung_Unten_Runter := FALSE;
	warten := FALSE;
END_IF

IF NOT Endl_Zufuehrer_Hinten THEN
	QZufuehrer_Antrieb_Rueck := TRUE;
ELSE 
	QZufuehrer_Antrieb_Rueck := FALSE;
END_IF
END_ACTION

ACTION Oben_Loesen_active:
QStammklemmung_Oben_Hoch := TRUE;
END_ACTION

ACTION Oben_Loesen_exit:
QStammklemmung_Oben_Hoch := FALSE;
END_ACTION

ACTION Pause_active:
Holz_Geklemmt := TRUE;
END_ACTION

ACTION Reset_active:
//Hydraulik
QStammklemmung_Oben_Hoch := 
QStammklemmung_Oben_Runter := 
QStammklemmung_Unten_Hoch := 
QStammklemmung_Unten_Runter := 
QSaege_Senken := 
QSaege_Heben := 
//Ausgänge Schalten
QHydraulikpumpe_EIN := 
QZufuehrer_Antrieb_vor := 
QZufuehrer_Antrieb_Rueck := 
QSaege_Antrieb_Ein := 
QKettenschmierung_EIN := 
Warten_Auf_Weiterschalten :=
Zyklus_Beendet := FALSE;

QHydraulikpumpe_EIN := TRUE;
END_ACTION

ACTION Saege_An_active:
QSaege_Antrieb_Ein := TRUE;
END_ACTION

ACTION Saege_Heben_active:
QSaege_Heben := TRUE;
END_ACTION

ACTION Saege_Heben_exit:
QSaege_Heben := FALSE;
QSaege_Antrieb_Ein := FALSE;
END_ACTION

ACTION Saegen_active:
QSaege_Senken := TRUE;
END_ACTION

ACTION Saegen_exit:
QSaege_Senken := FALSE;
END_ACTION

ACTION Unten_Loesen_active:
QStammklemmung_Unten_Runter := TRUE;
END_ACTION

ACTION Unten_Loesen_exit:
QStammklemmung_Unten_Runter := FALSE;
END_ACTION

ACTION von_oben_Klemmen_active:
QStammklemmung_Oben_Runter := TRUE;
END_ACTION

ACTION von_oben_Klemmen_exit:
QStammklemmung_Oben_Runter := FALSE;
END_ACTION

ACTION von_unten_Klemmen_active:
QStammklemmung_Unten_Hoch := TRUE;
END_ACTION

ACTION von_unten_Klemmen_exit:
QStammklemmung_Unten_Hoch := FALSE;
END_ACTION

ACTION VorPos_Saegen_entry:
Holz_Fertig := True;
END_ACTION

END_FUNCTION_BLOCK

// ---- POUs/Unterfunktionen/Meldeleuchte.TcPOU
FUNCTION_BLOCK Meldeleuchte
VAR_INPUT
	Zyklus_beendet : BOOL;
	Maschine_EIN : BOOL;
	Fehler_liegt_an : BOOL;
	Kettenschmierung_nicht_leer : BOOL;
	Busy : BOOL;
	Warten_auf_weiterschalten : BOOL;
	Warten_auf_Material : BOOL;
	Referenz_gefahren : BOOL;
	
END_VAR
VAR_OUTPUT
	OUT_Meldeleuchte_Rot AT %Q* : BOOL;//Rot Leuchten: Fehler, Rot Blinken: Kettenöl leer
	OUT_Meldeleuchte_Gelb AT %Q* : BOOL;//Gelb Leuchten:Referenz fehlt, Gelb Blinken: Zyklus beendet
	OUT_Meldeleuchte_Gruen AT %Q* : BOOL;//Grün Leuchten: Zyklus läuft, Grün Blinken: Zyklus läuft(warten auf weiterschalten)
	
END_VAR
VAR
	Impulsgeber : BLINK;
	TON_Timer_Impuls : TON;
	TON_Timer_Pause : TON;
	Impuls_Zeit : TIME := T#500MS;
	Pause_Zeit : TIME := T#500MS;
	Impuls : BOOL;
END_VAR

OUT_Meldeleuchte_Rot := OUT_Meldeleuchte_Gelb := OUT_Meldeleuchte_Gruen := FALSE;

Impulsgeber(
	ENABLE := TRUE,
	TIMELOW := Pause_Zeit,
	TIMEHIGH := Impuls_Zeit,
	OUT => Impuls);

IF Maschine_EIN AND NOT Referenz_gefahren THEN
	OUT_Meldeleuchte_Gelb := TRUE;
ELSIF Maschine_EIN AND Zyklus_beendet THEN
	OUT_Meldeleuchte_Gelb := Impuls;
END_IF

IF Maschine_EIN AND Fehler_liegt_an THEN
	OUT_Meldeleuchte_Rot := TRUE;
ELSIF Maschine_EIN AND NOT Fehler_liegt_an AND NOT Kettenschmierung_nicht_leer THEN
	OUT_Meldeleuchte_Rot := Impuls;
END_IF

IF Maschine_EIN AND Busy AND NOT Warten_auf_weiterschalten THEN 
	OUT_Meldeleuchte_Gruen := TRUE;
ELSIF Maschine_EIN AND Busy AND Warten_auf_weiterschalten THEN
	OUT_Meldeleuchte_Gruen := Impuls;
END_IF

END_FUNCTION_BLOCK

// ---- POUs/Grundfunktionen/OID200DatenLesen.TcPOU
FUNCTION_BLOCK OID200DatenLesen
VAR_INPUT
END_VAR
VAR_OUTPUT
	
	iOID200Dist_zu_Holz : UINT;
	OID200SchaltSignal : BOOL;
	
END_VAR
VAR
	
	ProzessDatenOID200 AT %I* : ARRAY[0..1] OF BYTE;
	ProzessdatenWortOID200 : WORD;
	
END_VAR

ProzessDatenWortOID200 := BYTE_TO_WORD(ProzessdatenOID200[1]) OR SHL(BYTE_TO_WORD(ProzessdatenOID200[0]), 8);
iOID200Dist_zu_Holz := WORD_TO_UINT(SHR(ProzessdatenWortOID200, 4));
OID200SchaltSignal := ProzessDatenOID200[1].0;

END_FUNCTION_BLOCK

// ---- POUs/Unterfunktionen/Ansteuerung_Ausgaenge.TcPOU
FUNCTION_BLOCK Ansteuerung_Ausgaenge
VAR_INPUT
	Saege_Hoch : BOOL;
	Saege_Runter : BOOL;
	Stammklemmung_Oben_Hoch : BOOL;
	Stammklemmung_Oben_Runter : BOOL;
	Stammklemmung_Unten_Hoch : BOOL;
	Stammklemmung_Unten_Runter : BOOL;
	Saege_EIN: BOOL;
	Zufuehrer_Vor : BOOL;
	Zufuehrer_Rueck : BOOL;
	endl_Zufuehrer_vorne : BOOL;
	endl_Zufuehrer_hinten : BOOL;
	endl_Zufuehrer_Vorpos : BOOL;
	endl_Stammklemmung_Oben_Oben : BOOL;
	endl_Stammklemmung_Oben_Unten : BOOL;
	endl_Stammklemmung_Unten_Oben : BOOL;
	endl_Stammklemmung_Unten_Unten : BOOL;
	endl_Saege_Oben : BOOL;
	endl_Saege_Unten : BOOL;
	kettenschmierung_EIN : BOOL;
	
END_VAR
VAR_OUTPUT
	OUT_Saege_Senken AT %Q* : BOOL;
	OUT_Saege_Heben AT %Q* : BOOL;
	OUT_Stammklemmung_Oben_Hoch AT %Q* : BOOL;
	OUT_Stammklemmung_Oben_Runter AT %Q* : BOOL;
	OUT_Stammklemmung_Unten_Hoch AT %Q* : BOOL;
	OUT_Stammklemmung_Unten_Runter AT %Q* : BOOL;
	OUT_Saege_EIN AT %Q* : BOOL;
	OUT_Zufuehrer_Antrieb_Vor AT %Q* : BOOL;
	OUT_Zufuehrer_Antrieb_Rueck AT %Q* : BOOL;
	OUT_Zufuehrer_Antrieb_Enable AT %Q* : BOOL;
	OUT_Kettenschmierung_EIN AT %Q* : BOOL;
END_VAR
VAR
	Saege : Hydr_Ventil;
	Stammklemmung_Oben : Hydr_Ventil;
	Stammklemmung_unten : Hydr_Ventil;
END_VAR


Saege(
	Funktion_A:= Saege_Hoch AND NOT endl_Saege_Oben, 
	Funktion_B:= Saege_Runter AND NOT endl_Saege_Unten, 
	Andere_Ventile_in_Ruhestellung:= Stammklemmung_Oben.Ruhestellung AND Stammklemmung_unten.Ruhestellung, 
	OUT_Spule_A=> OUT_Saege_Heben, 
	OUT_Spule_B=> OUT_Saege_Senken, 
	Status_Invalide=> , 
	Warte_auf_anderes_Ventil=> );

OUT_Saege_EIN := Saege_EIN;
OUT_Kettenschmierung_EIN := kettenschmierung_EIN;
	
Stammklemmung_Oben(
	Funktion_A:= Stammklemmung_Oben_Hoch AND NOT endl_Stammklemmung_Oben_Oben, 
	Funktion_B:= Stammklemmung_Oben_Runter AND NOT endl_Stammklemmung_Oben_Unten, 
	Andere_Ventile_in_Ruhestellung:= Saege.Ruhestellung AND Stammklemmung_unten.Ruhestellung, 
	OUT_Spule_A=> OUT_Stammklemmung_Oben_Hoch, 
	OUT_Spule_B=> OUT_Stammklemmung_Oben_Runter, 
	Status_Invalide=> , 
	Warte_auf_anderes_Ventil=> );
	
Stammklemmung_unten(
	Funktion_A:= Stammklemmung_Unten_Hoch AND NOT endl_Stammklemmung_Unten_Oben, 
	Funktion_B:= Stammklemmung_Unten_Runter AND NOT endl_Stammklemmung_Unten_Unten, 
	Andere_Ventile_in_Ruhestellung:= Saege.Ruhestellung AND Stammklemmung_Oben.Ruhestellung, 
	OUT_Spule_A=> OUT_Stammklemmung_Unten_Hoch, 
	OUT_Spule_B=> OUT_Stammklemmung_Unten_Runter, 
	Status_Invalide=> ,  
	Warte_auf_anderes_Ventil=> );
	
OUT_Zufuehrer_Antrieb_Vor := Zufuehrer_Vor AND NOT Zufuehrer_Rueck AND NOT endl_Zufuehrer_vorne;
OUT_Zufuehrer_Antrieb_Rueck := Zufuehrer_Rueck AND NOT Zufuehrer_Vor AND NOT endl_Zufuehrer_hinten;
OUT_Zufuehrer_Antrieb_Enable := OUT_Zufuehrer_Antrieb_Vor OR OUT_Zufuehrer_Antrieb_Rueck;

END_FUNCTION_BLOCK

// ---- POUs/Grundfunktionen/Hydr_Ventil.TcPOU
FUNCTION_BLOCK Hydr_Ventil
VAR_INPUT
	Funktion_A : BOOL;
	Funktion_B : BOOL;
	Andere_Ventile_in_Ruhestellung : BOOL;
END_VAR
VAR_OUTPUT
	OUT_Spule_A : BOOL;
	OUT_Spule_B : BOOL;
	Status_Invalide : BOOL;
	Ruhestellung : BOOL;
	Warte_auf_anderes_Ventil : BOOL;
END_VAR
VAR
END_VAR


IF Funktion_A AND NOT Funktion_B AND Andere_Ventile_in_Ruhestellung THEN 
	OUT_Spule_A := TRUE;
ELSIF NOT Funktion_A THEN 
	OUT_Spule_A := FALSE;
END_IF

IF Funktion_B AND NOT Funktion_A AND Andere_Ventile_in_Ruhestellung THEN
	OUT_Spule_B := TRUE;
ELSIF NOT Funktion_B THEN 
	OUT_Spule_B := FALSE;
END_IF

Status_Invalide := Funktion_A AND Funktion_B;
Ruhestellung := NOT OUT_Spule_A AND NOT OUT_Spule_B;
Warte_auf_anderes_Ventil := Funktion_A OR Funktion_B AND NOT Andere_Ventile_in_Ruhestellung;

END_FUNCTION_BLOCK

// ---- GlobalTextList.TcGTLO
TEXTLIST GlobalTextList
  773 = 'A'
  944 = 'Autoatikbetrieb'
  601 = 'Hydraulik EIN'
  473 = 'Kein Notaus'
  194 = 'M'
  891 = 'Manueller Betrieb'
  390 = 'Maschine EIN'
  28 = 'R'
  320 = 'Referenzfahrt'
  216 = 'Text'
  214 = 'W'
  30 = 'Warmlauf'
  904 = 'Zyklus Start'
  281 = 'Zyklus Stopp'
END_TEXTLIST

// ---- VISUs/Visualization.TcVIS
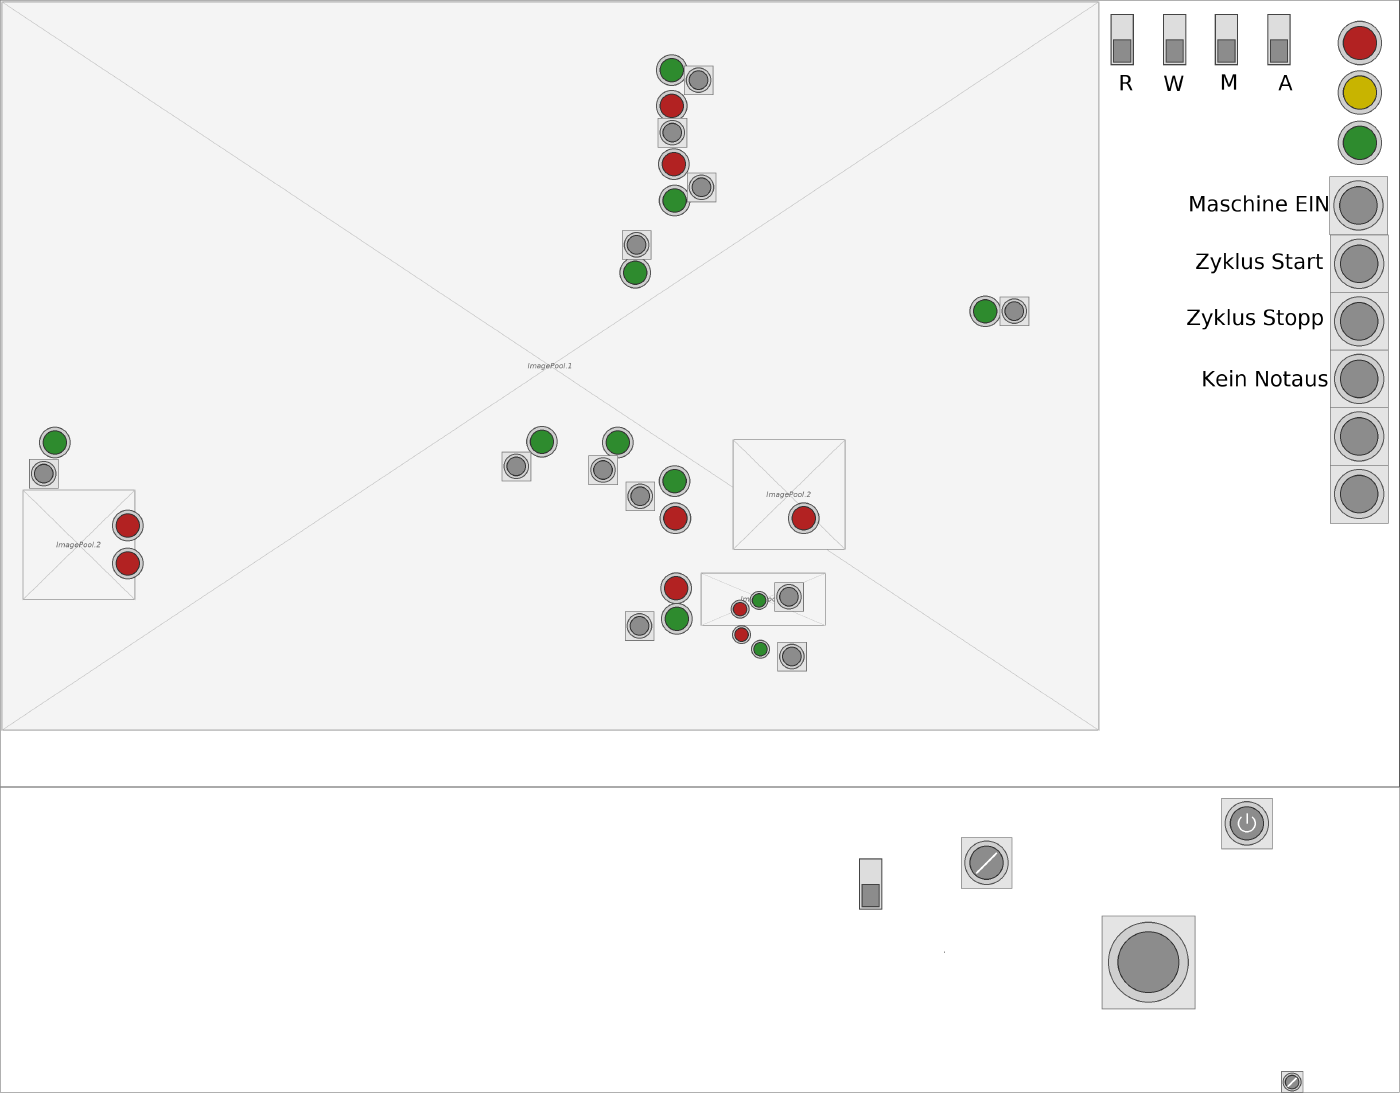
VISUALIZATION Visualization  // 1920x1500
    Rectangle (0,0 1920x1080)
    Image (2,2 1505x1000), image: ImagePool.1
    Image (1005,603 154x151), angle 26, image: ImagePool.2
    Image (31,672 154x151), image: ImagePool.2
    Lamp1 (1077,686 50x50), variable: MAIN.Saegeautomat.Ansteuerung_Ausgaenge.OUT_Saege_EIN, style: Lamp-Lamp1-Red
    Lamp1 (150,696 50x50), variable: MAIN.Saegeautomat.Ansteuerung_Ausgaenge.OUT_Zufuehrer_Antrieb_Vor, style: Lamp-Lamp1-Red
    Lamp1 (150,748 50x50), variable: MAIN.Saegeautomat.Ansteuerung_Ausgaenge.OUT_Zufuehrer_Antrieb_Rueck, style: Lamp-Lamp1-Red
    Lamp1 (1326,402 50x50), variable: MAIN.Saegeautomat.IN_Schaltausg_Lichtschranke, style: Lamp-Lamp1-Green
    Lamp1 (900,635 50x50), variable: MAIN.Saegeautomat.IN_Endl_Untere_Stammklemmung_Oben, style: Lamp-Lamp1-Green
    Lamp1 (903,824 50x50), variable: MAIN.Saegeautomat.IN_Endl_Untere_Stammklemmung_Unten, style: Lamp-Lamp1-Green
    Lamp1 (900,250 50x50), variable: MAIN.Saegeautomat.IN_Endl_Obere_Stammklemmung_Unten, style: Lamp-Lamp1-Green
    Lamp1 (896,71 50x50), variable: MAIN.Saegeautomat.IN_Endl_Obere_Stammklemmung_Oben, style: Lamp-Lamp1-Green
    Lamp1 (846,349 50x50), variable: MAIN.Saegeautomat.IN_Endl_Tastschiene, style: Lamp-Lamp1-Green
    Lamp1 (822,582 50x50), variable: MAIN.Saegeautomat.IN_Endl_Zufuehrer_Vorne, style: Lamp-Lamp1-Green
    Lamp1 (718,581 50x50), variable: MAIN.Saegeautomat.IN_Vorposition_Zufuehrer, style: Lamp-Lamp1-Green
    Lamp1 (50,582 50x50), variable: MAIN.Saegeautomat.IN_Endl_Zufuehrer_Hinten, style: Lamp-Lamp1-Green
    Image (961,786 171x72), angle 97, image: ImagePool.3
    Lamp1 (1028,876 30x30), variable: MAIN.Saegeautomat.IN_Endl_Saege_Oben, style: Lamp-Lamp1-Green
    Lamp1 (1026,809 30x30), variable: MAIN.Saegeautomat.IN_Endl_Saege_Unten, style: Lamp-Lamp1-Green
    Lamp1 (901,686 50x50), variable: MAIN.Saegeautomat.Ansteuerung_Ausgaenge.OUT_Stammklemmung_Unten_Hoch, style: Lamp-Lamp1-Red
    Lamp1 (902,782 50x50), variable: MAIN.Saegeautomat.Ansteuerung_Ausgaenge.OUT_Stammklemmung_Unten_Runter, style: Lamp-Lamp1-Red
    Lamp1 (899,200 50x50), variable: MAIN.Saegeautomat.Ansteuerung_Ausgaenge.OUT_Stammklemmung_Oben_Runter, style: Lamp-Lamp1-Red
    Lamp1 (896,120 50x50), variable: MAIN.Saegeautomat.Ansteuerung_Ausgaenge.OUT_Stammklemmung_Oben_Hoch, style: Lamp-Lamp1-Red
    Lamp1 (1000,821 30x30), variable: MAIN.Saegeautomat.Ansteuerung_Ausgaenge.OUT_Saege_Senken, style: Lamp-Lamp1-Red
    Lamp1 (1002,856 30x30), variable: MAIN.Saegeautomat.Ansteuerung_Ausgaenge.OUT_Saege_Heben, style: Lamp-Lamp1-Red
    RotarySwitch (1318,1149 70x70), behaviour: TOGGLE, style: Switch-RotarySwitch-Gray
    PushSwitch (1824,322 80x80), variable: MAIN.Saegeautomat.IN_Zyklus_Start, behaviour: TAP, style: Switch-PushSwitch-Gray
    PushSwitchLed (1293,1306 4x1), behaviour: TOGGLE, style: Switch-PushSwitchLed-Gray
    PushSwitchLed (1511,1254 128x133), behaviour: TOGGLE, style: Switch-PushSwitchLed-Gray
    DipSwitch (1159,1178 70x70), behaviour: TOGGLE, style: Switch-DipSwitch-Gray
    Lamp1 (1830,24 70x70), variable: MAIN.Saegeautomat.Steuerung_Meldeleuchten.OUT_Meldeleuchte_Rot, style: Lamp-Lamp1-Red
    Lamp1 (1830,92 70x70), variable: MAIN.Saegeautomat.Steuerung_Meldeleuchten.OUT_Meldeleuchte_Gelb, style: Lamp-Lamp1-Yellow
    Lamp1 (1830,161 70x70), variable: MAIN.Saegeautomat.Steuerung_Meldeleuchten.OUT_Meldeleuchte_Gruen, style: Lamp-Lamp1-Green
    PushSwitch (1824,401 80x80), variable: MAIN.Saegeautomat.IN_Zyklus_Stopp, behaviour: TAP, style: Switch-PushSwitch-Gray
    PushSwitch (1824,480 80x80), variable: MAIN.Saegeautomat.IN_Kein_Notaus, behaviour: TOGGLE, style: Switch-PushSwitch-Gray
    PushSwitch (1824,559 80x80), behaviour: TOGGLE, style: Switch-PushSwitch-Gray
    PushSwitch (1824,638 80x80), behaviour: TOGGLE, style: Switch-PushSwitch-Gray
    PushSwitch (1823,242 80x80), variable: MAIN.Saegeautomat.IN_Maschine_EIN, behaviour: TAP, style: Switch-PushSwitch-Gray
    PowerSwitch (1675,1095 70x70), behaviour: TOGGLE, style: Switch-PowerSwitch-Gray
    RotarySwitch (1697,1470 150x30), behaviour: TOGGLE, style: Switch-RotarySwitch-Gray
    DipSwitch (1719,19 70x70), variable: MAIN.Saegeautomat.IN_BetriebsArt_Automatik, behaviour: TOGGLE, style: Switch-DipSwitch-Gray
    DipSwitch (1647,19 70x70), variable: MAIN.Saegeautomat.IN_BetriebsArt_Manuell, behaviour: TOGGLE, style: Switch-DipSwitch-Gray
    DipSwitch (1504,19 70x70), variable: MAIN.Saegeautomat.IN_BetriebsArt_Referenz, behaviour: TOGGLE, style: Switch-DipSwitch-Gray
    DipSwitch (1576,19 70x70), variable: MAIN.Saegeautomat.IN_BetriebsArt_Warmlauf, behaviour: TOGGLE, style: Switch-DipSwitch-Gray
    Label (1583,344 235x30), "Zyklus Start"
    Label (1584,421 235x30), "Zyklus Stopp"
    Label (1590,505 235x30), "Kein Notaus"
    Label (1592,265 235x30), "Maschine EIN"
    Label (1517,99 40x30), "R"
    Label (1587,100 40x30), "W"
    Label (1661,98 40x30), "M"
    Label (1736,99 40x30), "A"
    PushSwitch (1062,799 40x40), variable: MAIN.Saegeautomat.IN_Endl_Saege_Unten, behaviour: TOGGLE, style: Switch-PushSwitch-Gray
    PushSwitch (1066,881 40x40), variable: MAIN.Saegeautomat.IN_Endl_Saege_Oben, behaviour: TOGGLE, style: Switch-PushSwitch-Gray
    PushSwitch (857,839 40x40), variable: MAIN.Saegeautomat.IN_Endl_Untere_Stammklemmung_Unten, behaviour: TOGGLE, style: Switch-PushSwitch-Gray
    PushSwitch (858,661 40x40), variable: MAIN.Saegeautomat.IN_Endl_Untere_Stammklemmung_Oben, behaviour: TOGGLE, style: Switch-PushSwitch-Gray
    PushSwitch (807,625 40x40), variable: MAIN.Saegeautomat.IN_Endl_Zufuehrer_Vorne, behaviour: TOGGLE, style: Switch-PushSwitch-Gray
    PushSwitch (688,620 40x40), variable: MAIN.Saegeautomat.IN_Vorposition_Zufuehrer, behaviour: TOGGLE, style: Switch-PushSwitch-Gray
    PushSwitch (40,630 40x40), variable: MAIN.Saegeautomat.IN_Endl_Zufuehrer_Hinten, behaviour: TOGGLE, style: Switch-PushSwitch-Gray
    PushSwitch (853,316 40x40), variable: MAIN.Saegeautomat.IN_Endl_Tastschiene, behaviour: TOGGLE, style: Switch-PushSwitch-Gray
    PushSwitch (942,237 40x40), variable: MAIN.Saegeautomat.IN_Endl_Obere_Stammklemmung_Unten, behaviour: TOGGLE, style: Switch-PushSwitch-Gray
    PushSwitch (938,90 40x40), variable: MAIN.Saegeautomat.IN_Endl_Obere_Stammklemmung_Oben, behaviour: TOGGLE, style: Switch-PushSwitch-Gray
    PushSwitch (1371,407 40x40), variable: MAIN.Saegeautomat.IN_Schaltausg_Lichtschranke, behaviour: TOGGLE, style: Switch-PushSwitch-Gray
    PushSwitch (902,162 40x40), variable: MAIN.Saegeautomat.IN_Schaltausg_Druckschalter_Obere_Klemmung, behaviour: TOGGLE, style: Switch-PushSwitch-Gray
END_VISUALIZATION
